// TwinCAT 3 PLC project StateMachinePractice
// ProgramVersion: 3.1.4024.0
// libraries:
//   Tc2_Standard, * (Beckhoff Automation GmbH)
//   Tc2_System, * (Beckhoff Automation GmbH)
//   Tc3_Module, * (Beckhoff Automation GmbH)
// project tree:
//   DUTs/ E_MachineState.TcDUT
//   / PlcTask.TcTTO
//   POUs/ FB_Drill.TcPOU, MAIN.TcPOU
// (motion and I/O tree: see PLC project functionblockpractice)
// real-time tasks:
//   TASK PlcTask: cycle T#10ms, priority 20, ADS port 350
//   TASK PlcTask2: cycle T#10ms, priority 22, ADS port 352
//   TASK PlcTask1: cycle T#10ms, priority 21, ADS port 351
//   TASK PlcTask3: cycle T#10ms, priority 23, ADS port 353
//   TASK PlcTask4: cycle T#10ms, priority 24, ADS port 354
//   TASK PlcTask5: cycle T#10ms, priority 25, ADS port 355
//   TASK PlcTask6: cycle T#10ms, priority 26, ADS port 356

CONFIGURATION StateMachinePractice
    RESOURCE PLC ON TwinCAT3
        TASK PlcTask(INTERVAL := T#10ms, PRIORITY := 26);
        PROGRAM MAIN WITH PlcTask : MAIN;
    END_RESOURCE
END_CONFIGURATION

// ---- DUTs/E_MachineState.TcDUT
{attribute 'qualified_only'}
{attribute 'strict'}
TYPE E_MachineState :
(
	IDLE := 0,
	Drilling,
	Retracting,
	Error
);
END_TYPE

// ---- POUs/MAIN.TcPOU
PROGRAM MAIN
VAR
	eState : E_MachineState;
	bStart : BOOL;
	bLimitUp : BOOL;
	bLimitDown : BOOL;
	bEmergencyStop : BOOL;
	bDrilling : BOOL;
	bRetracting : BOOL;
	
	
END_VAR


IF bEmergencyStop THEN
	 eState := E_MachineState.Error;
END_IF

CASE eState OF
	E_MachineState.IDLE :
	bDrilling := FALSE;
	bRetracting := FALSE;
	IF MAIN.TRANS_DrillCheck THEN
		eState := E_MachineState.Drilling;
	END_IF
	
	E_MachineState.Drilling :
	bDrilling := TRUE;
	bRetracting := FALSE;
	bLimitUp := FALSE;
	IF bStart AND bLimitDown THEN
		eState := E_MachineState.Retracting;
	END_IF
	
	E_MachineState.Retracting :
	bDrilling := FALSE;
	bRetracting := TRUE;
	bLimitDown := FALSE;
	IF bStart AND bLimitUp THEN
		eState := E_MachineState.IDLE;
	END_IF
	
	E_MachineState.Error :
	bDrilling := FALSE;
	bRetracting := FALSE;
	IF  NOT bEmergencyStop AND bStart THEN
		eState := E_MachineState.IDLE;
	END_IF
	
	
END_CASE

TRANSITION TRANS_DrillCheck:
TRANS_DrillCheck := (bStart AND bLimitUp);
END_TRANSITION

END_PROGRAM

// ---- POUs/FB_Drill.TcPOU
FUNCTION_BLOCK FB_Drill
VAR_INPUT
	bStart : BOOL;
END_VAR
VAR_OUTPUT
END_VAR
VAR
END_VAR

TRANSITION TRANS_Check:
TRANS_Check := bStart;
END_TRANSITION

END_FUNCTION_BLOCK
